TYPE Str_fb_mem :
STRUCT
	State : E_State_PackML;
END_STRUCT
END_TYPE

(* stored: Version 1.1.0.1, ProductVersion 3.1.4024.12
   DUT Str_fb_mem: Id {91f2edbf-eab2-4cf1-90d4-b3264c4a9188} *)
